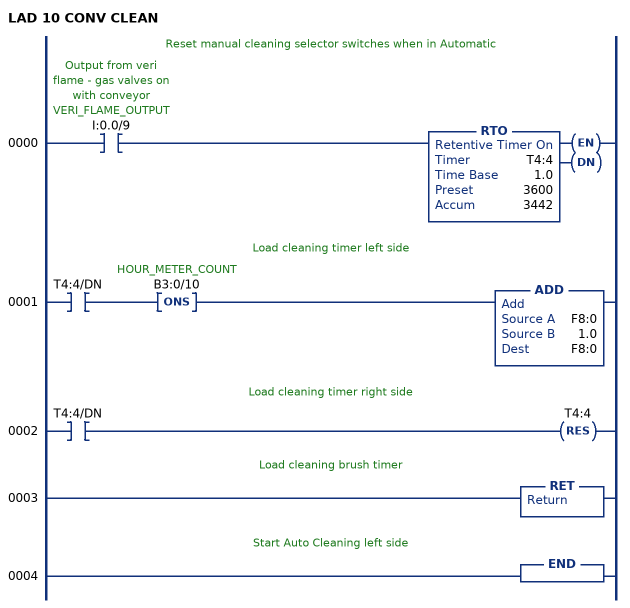
% Rung: 0 %
% Reset manual cleaning selector switches when in Automatic %
SOR XIC I:0.0/9 RTO T4:4 1.0 3600 3442 EOR
%   I:0.0/9  VERI_FLAME_OUTPUT  "Output from veri flame - gas valves on with conveyor" %
% Rung: 1 %
% Load cleaning timer left side %
SOR XIC T4:4/DN ONS B3:0/10 ADD F8:0 1.0 F8:0 EOR
%   B3:0/10  HOUR_METER_COUNT %
% Rung: 2 %
% Load cleaning timer right side %
SOR XIC T4:4/DN RES T4:4 EOR
% Rung: 3 %
% Load cleaning brush timer %
SOR RET EOR
% Rung: 4 %
% Start Auto Cleaning left side %
SOR END EOR

LADDER 11 "FAULTS"
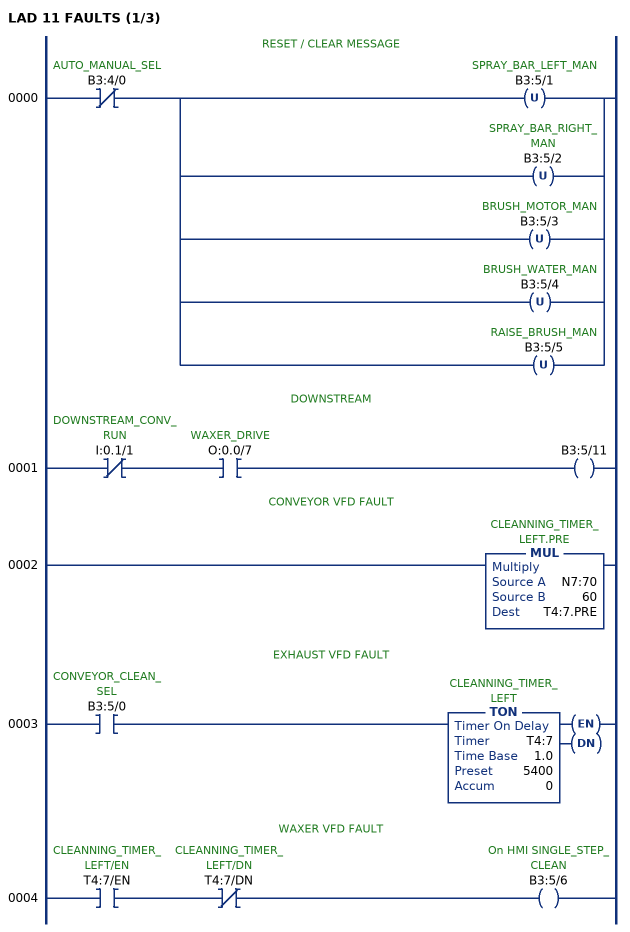
% Rung: 0 %
% RESET / CLEAR MESSAGE %
SOR XIO B3:4/0 BST OTU B3:5/1 NXB BST OTU B3:5/2 NXB BST OTU B3:5/3 NXB BST OTU B3:5/4 NXB OTU B3:5/5 BND BND BND BND EOR
%   B3:4/0  AUTO_MANUAL_SEL %
%   B3:5/1  SPRAY_BAR_LEFT_MAN %
%   B3:5/2  SPRAY_BAR_RIGHT_MAN %
%   B3:5/3  BRUSH_MOTOR_MAN %
%   B3:5/4  BRUSH_WATER_MAN %
%   B3:5/5  RAISE_BRUSH_MAN %
% Rung: 1 %
% DOWNSTREAM %
SOR XIO I:0.1/1 XIC O:0.0/7 OTE B3:5/11 EOR
%   I:0.1/1  DOWNSTREAM_CONV_RUN %
%   O:0.0/7  WAXER_DRIVE %
% Rung: 2 %
% CONVEYOR VFD FAULT %
SOR MUL N7:70 60 T4:7.PRE EOR
%   N7:70  CLEANING_TIME_LEFT %
%   T4:7  CLEANNING_TIMER_LEFT %
% Rung: 3 %
% EXHAUST VFD FAULT %
SOR XIC B3:5/0 TON T4:7 1.0 5400 0 EOR
%   B3:5/0  CONVEYOR_CLEAN_SEL %
%   T4:7  CLEANNING_TIMER_LEFT %
% Rung: 4 %
% WAXER VFD FAULT %
SOR XIC T4:7/EN XIO T4:7/DN OTE B3:5/6 EOR
%   T4:7  CLEANNING_TIMER_LEFT %
%   B3:5/6  SINGLE_STEP_CLEAN  "On HMI" %

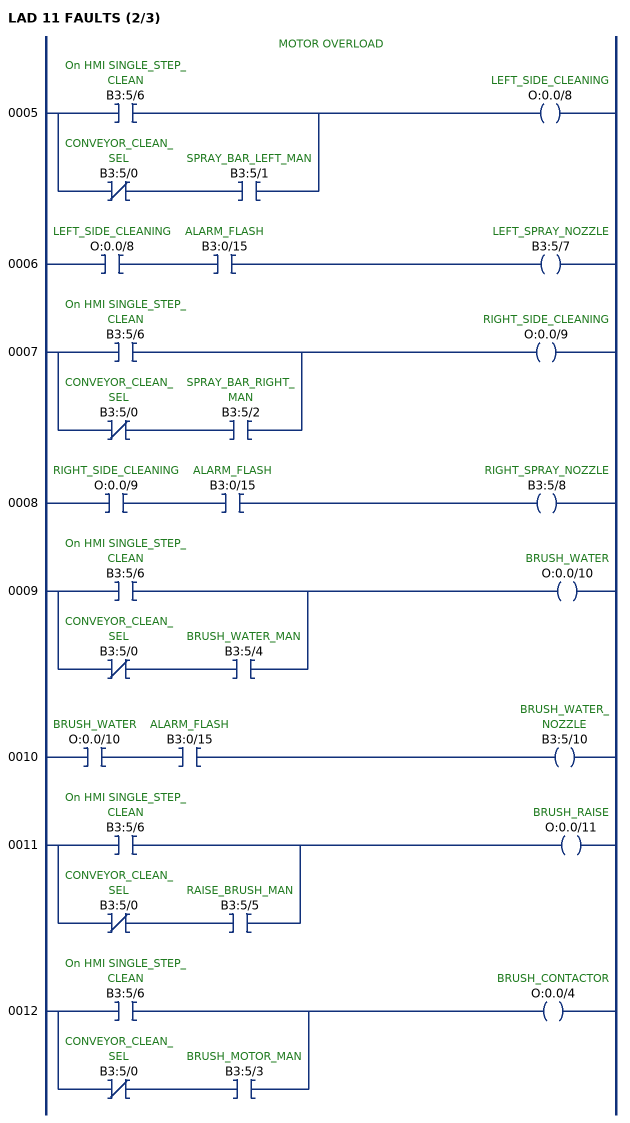
% Rung: 5 %
% MOTOR OVERLOAD %
SOR BST XIC B3:5/6 NXB XIO B3:5/0 XIC B3:5/1 BND OTE O:0.0/8 EOR
%   B3:5/6  SINGLE_STEP_CLEAN  "On HMI" %
%   B3:5/0  CONVEYOR_CLEAN_SEL %
%   B3:5/1  SPRAY_BAR_LEFT_MAN %
%   O:0.0/8  LEFT_SIDE_CLEANING %
% Rung: 6 %
SOR XIC O:0.0/8 XIC B3:0/15 OTE B3:5/7 EOR
%   O:0.0/8  LEFT_SIDE_CLEANING %
%   B3:0/15  ALARM_FLASH %
%   B3:5/7  LEFT_SPRAY_NOZZLE %
% Rung: 7 %
SOR BST XIC B3:5/6 NXB XIO B3:5/0 XIC B3:5/2 BND OTE O:0.0/9 EOR
%   B3:5/6  SINGLE_STEP_CLEAN  "On HMI" %
%   B3:5/0  CONVEYOR_CLEAN_SEL %
%   B3:5/2  SPRAY_BAR_RIGHT_MAN %
%   O:0.0/9  RIGHT_SIDE_CLEANING %
% Rung: 8 %
SOR XIC O:0.0/9 XIC B3:0/15 OTE B3:5/8 EOR
%   O:0.0/9  RIGHT_SIDE_CLEANING %
%   B3:0/15  ALARM_FLASH %
%   B3:5/8  RIGHT_SPRAY_NOZZLE %
% Rung: 9 %
SOR BST XIC B3:5/6 NXB XIO B3:5/0 XIC B3:5/4 BND OTE O:0.0/10 EOR
%   B3:5/6  SINGLE_STEP_CLEAN  "On HMI" %
%   B3:5/0  CONVEYOR_CLEAN_SEL %
%   B3:5/4  BRUSH_WATER_MAN %
%   O:0.0/10  BRUSH_WATER %
% Rung: 10 %
SOR XIC O:0.0/10 XIC B3:0/15 OTE B3:5/10 EOR
%   O:0.0/10  BRUSH_WATER %
%   B3:0/15  ALARM_FLASH %
%   B3:5/10  BRUSH_WATER_NOZZLE %
% Rung: 11 %
SOR BST XIC B3:5/6 NXB XIO B3:5/0 XIC B3:5/5 BND OTE O:0.0/11 EOR
%   B3:5/6  SINGLE_STEP_CLEAN  "On HMI" %
%   B3:5/0  CONVEYOR_CLEAN_SEL %
%   B3:5/5  RAISE_BRUSH_MAN %
%   O:0.0/11  BRUSH_RAISE %
% Rung: 12 %
SOR BST XIC B3:5/6 NXB XIO B3:5/0 XIC B3:5/3 BND OTE O:0.0/4 EOR
%   B3:5/6  SINGLE_STEP_CLEAN  "On HMI" %
%   B3:5/0  CONVEYOR_CLEAN_SEL %
%   B3:5/3  BRUSH_MOTOR_MAN %
%   O:0.0/4  BRUSH_CONTACTOR %

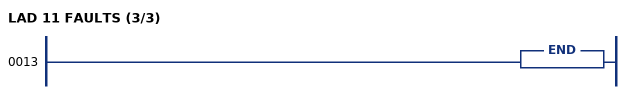
% Rung: 13 %
SOR END EOR

OTHER DOCUMENTED ADDRESSES
  B3:0/11  FLAME_STANDBY
  B3:0/14  SET_MIN_VFD_SPEED
  B3:1/8  IN_8  "High Temp Limit"
  B3:2/8  FE_HIGH_TEMP_LIMIT  "Fault Enable"
  B3:3/8  FC_HIGH_TEMP_LIMIT  "Fault Catch"
  B3:4/7  PILOT_VALVE_OPEN
  B3:4/8  PILOT_VALVE_CLOSED
  B3:4/13  DISPLAY_CNT_DN_TIME
  B3:5/13  WAXER_DRIVE_SEL
  B3:5/15  POP_UP_SCREEN  "On HMI"
  I:0.0/10  DRYER_CONVEYOR_AUX1  "Valve Train to gas valve"
  I:0.0/11  VERI_FLAME_PILOT
  I:0.0/12  VERI_FLAME_IGNITION
  I:0.0/14  VALVE_PROVING_ALARM
  I:0.1/3  CONV_VFD_FAULT
  I:0.1/4  EXHAUST_VFD_FAULT
  I:0.1/5  WAXER_VFD_FAULT
  I:0.1/6  WAXER_RUNNING
  I:1.0/0  TC1
  I:2.0/0  SENSOR_PLENUM
  I:2.0/1  SENSOR_RETURN
  I:2.1/0  SENSOR_Q
  I:2.2/0  SENSOR_HUMIDITY
  I:2.3/0  SENSOR_TEMP_RHL
  N7:23  ADVERAGE_OF_1_2_3
  N7:30  PV_RH_PROCESS_VAR  "Feedback from humidity sensors - calculated value"
  N7:46  PLENUM_PS_ALARM
  N7:59  SCALLED_SPEED_REF
  N7:63  TEMP_SET_POINT  "For conveyor start"
  N7:65  FAULT_MESSAGES
  N7:66  CONV_SPEED_SCALLER
  N7:67  CONVEYOR_SPEED
  N7:71  CLEANING_TIME_RIGHT
  N7:72  CLEANING_TIME_BRUSH
  O:0.0/3  LUB_SOLENOID
  PD9:0.3  "SPS Setpoint"
  PFILE:5  "a"
  PFILE:10  "Brush Clening"
  T4:8  CLEANING_TIMER_RIGHT
  T4:9  CLEANING_TIMER_BRUSH

COMMENTS NOT ATTACHED TO A CURRENT RUNG
  N7:3: Subract to bring sensor value to zero
  N7:65: CONVEYOR VFD FAULT
  N7:53: Find slope intercept  b value step #2 -  multiply point Ax times slope
  N7:52: Multiply RH difference by Speed Scaller
  N7:50: Find slope step #2 -  multiply Y dif by 100 to get better accuracy
  N7:56: Solve for speed Step #2 - divide by 100 (multiply slope times humidity)
  N7:55: Find slope intercept  b value step #5 -  sub Ay minus Ax*slope
  N7:54: Find slope intercept  b value step #3 -  multiply point Ay by 100 for Accuracy
  N7:0: Read input card - Return Pressure
  RUNG000010-000005: Start Auto Cleaning left side
  RUNG000010-000006: Start Auto Cleaning left side
  RUNG000010-000007: Manual and Automatic cleaning function select
  RUNG000010-000009: Manual and Automatic cleaning function select
  RUNG000010-000011: Manual and Automatic cleaning function select
  RUNG000010-000013: Manual and Automatic cleaning function select
  RUNG000010-000014: Manual and Automatic cleaning function select

DATA TABLE (non-zero values as saved)
DATA B3
% B3:0 % 0X8290 0X8000 0X0000 0X0000 0X0180 0X0000 0X0000 0X0102 0X0000 0X0000
% B3:10 % 0X0001 0X0000 0X0000 0X0000 0X0000 0X0000 0X0000 0X0000 0X0000 0X0000
DATA T4
% .PRE .ACC %
% T4:0 % 1799 0
% T4:1 % 1 0
% T4:2 % 150 150
% T4:3 % 100 12
% T4:4 % 3600 3442
% T4:5 % 60 0
% T4:6 % 4 4
% T4:7 % 5400 0
% T4:8 % 600 0
% T4:9 % 1800 0
% T4:10 % 9999 0
DATA N7
% N7:0 % 8183 6226 105 1 19 6226 6265 18 1 -2
% N7:10 % 233 230 225 683 200 1400 1200 683 16383 3400
% N7:20 % 20738 6250 240 10 139 25 25 50 100 12
% N7:30 % 10 0 195 9776 16277 30 1799 68 14 120
% N7:40 % 2 5 3 200 0 5 0 0 0 1200
% N7:50 % 0 10 0 0 60 2 20 20 0 0
% N7:60 % 60 0 0 0 0 0 0 0 0 0
% N7:70 % 90 0 0 0 0 0 0
DATA F8
% F8:0 % 303
